PROGRAM MAIN
VAR
END_VAR

PRG_Safe();

END_PROGRAM

(* stored: Version 1.1.0.1, ProductVersion 3.1.4024.9
   POU MAIN: Id {f5b8053c-ab5a-49d4-b365-7b1c9572599e}, SpecialFunc None *)
